Fanuc KAREL source: kd00062.KL

-- PROVISIONAL review KL for V1013-1; original PC SHA256 eb705cf7d7deba4f51a17e7931a45f1b3af2ed2da5167265dff379eb69365117
-- Incomplete behavior may be omitted. Consult companion uncertainty JSON. Do not deploy.
PROGRAM KD00062
%NOLOCKGROUP
VAR
  I : INTEGER
  J : INTEGER
  B : BOOLEAN
  R : REAL
  S : STRING[80]
BEGIN
  -- UNRESOLVED_PC offsets 5-18; opcodes 9D,81,18,9D,1B,9D,12,9D,13,04
  -- UNRESOLVED_PC offsets 23-27; opcodes 7F
END KD00062
